Omron CX-Programmer project NewProject (CX-Programmer 7.21)

# PLC NewPLC1: CJ1M CPU13
I/O table (CPU CJ1M-CPU13): rack 0 slot 0 CJ1W-SCU41-V1

## Global symbols (name address type ; comment)
D0 CHANNEL  ; Ctrl1
D1 CHANNEL  ; Ctrl2
D10 CHANNEL  ; Send Word
D20 CHANNEL  ; No. To Send
D30 CHANNEL  ; Receive Word
D40 CHANNEL  ; No. To Receive
D70 CHANNEL  ; Batt
D71 CHANNEL  ; Sgn1
D72 CHANNEL  ; Dig1
D73 CHANNEL  ; Sgn2
D74 CHANNEL  ; Dig2
D75 CHANNEL  ; ID
D76 CHANNEL  ; Disp1
D77 CHANNEL  ; Dly
D78 CHANNEL  ; StpSgn
D79 CHANNEL  ; RunSgn
D80 CHANNEL  ; FinSgn
D81 CHANNEL  ; RsdSgn
D82 CHANNEL  ; Disp2
D83 CHANNEL  ; Err
D84 CHANNEL  ; Page
D85 CHANNEL  ; FileNo.
D86 CHANNEL  ; ErrNo.
D87 CHANNEL  ; DataNo.2
D88 CHANNEL  ; DataNo.1 LSB
D89 CHANNEL  ; MsdErr
D90 CHANNEL  ; MemSgn
D92 CHANNEL  ; DataNo.2 MSB
D93 CHANNEL  ; DataNo.

## Program NewProgram1 (cyclic task 0)

### Section Section1

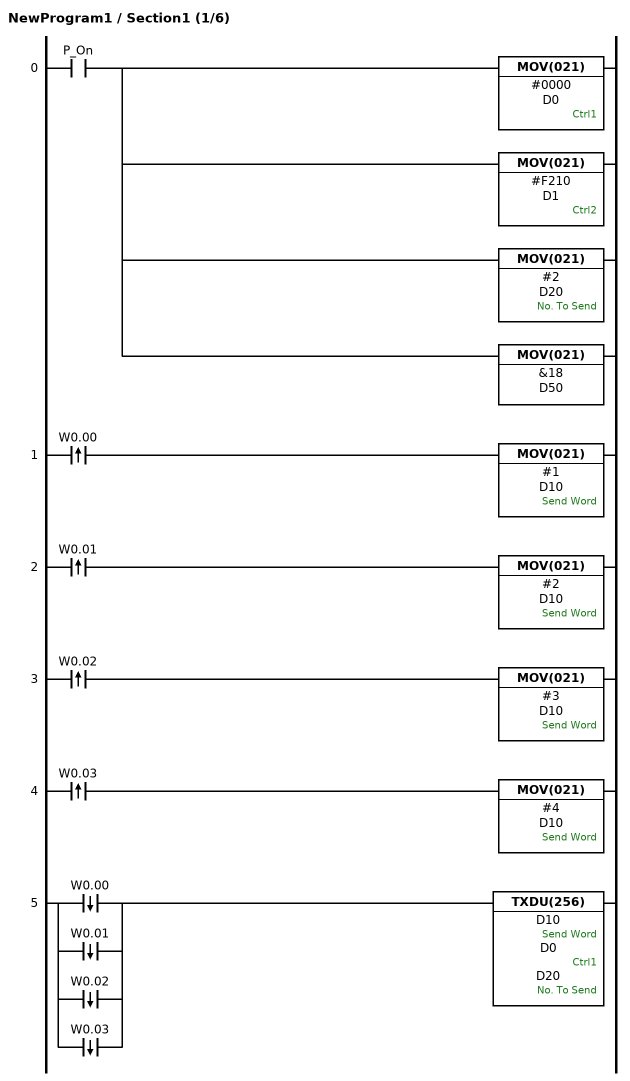
; rung 0
LD P_On
MOV(021) #0000 D0  ; Ctrl1
MOV(021) #F210 D1  ; Ctrl2
MOV(021) #2 D20  ; No. To Send
MOV(021) &18 D50
; rung 1
@LD W0.00
MOV(021) #1 D10  ; Send Word
; rung 2
@LD W0.01
MOV(021) #2 D10  ; Send Word
; rung 3
@LD W0.02
MOV(021) #3 D10  ; Send Word
; rung 4
@LD W0.03
MOV(021) #4 D10  ; Send Word
; rung 5
%LD W0.00
%OR W0.01
%OR W0.02
%OR W0.03
TXDU(256) D10 D0 D20  ; Send Word, Ctrl1, No. To Send

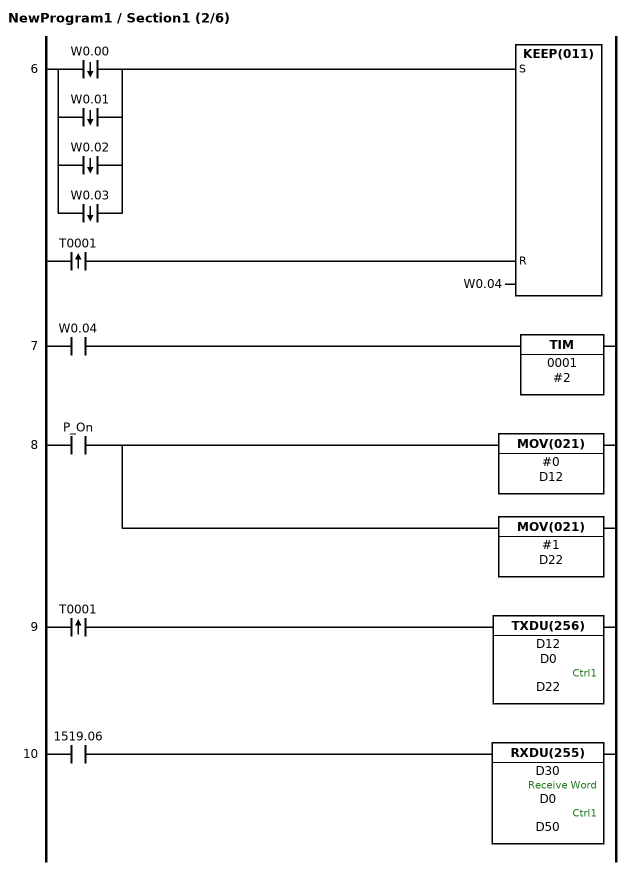
; rung 6
%LD W0.00
%OR W0.01
%OR W0.02
%OR W0.03
@LD T0001
KEEP(011) W0.04
; rung 7
LD W0.04
TIM 0001 #2
; rung 8
LD P_On
MOV(021) #0 D12
MOV(021) #1 D22
; rung 9
@LD T0001
TXDU(256) D12 D0 D22  ; Ctrl1
; rung 10
LD 1519.06
RXDU(255) D30 D0 D50  ; Receive Word, Ctrl1

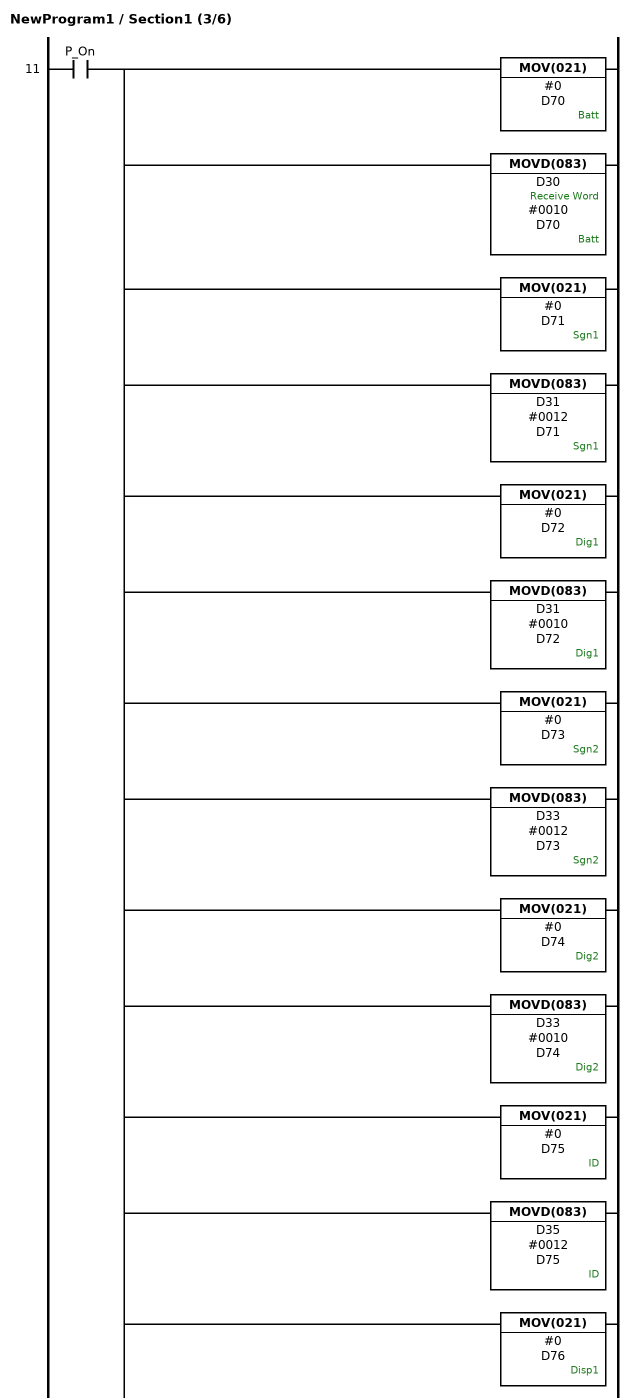

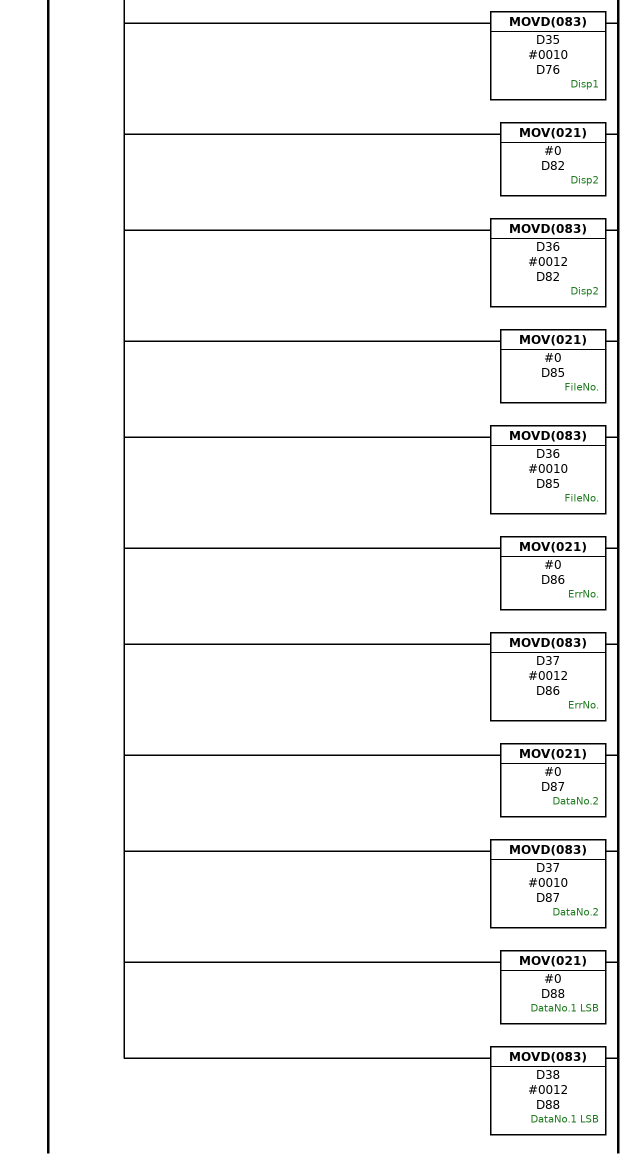
; rung 11
LD P_On
MOV(021) #0 D70  ; Batt
MOVD(083) D30 #0010 D70  ; Receive Word, Batt
MOV(021) #0 D71  ; Sgn1
MOVD(083) D31 #0012 D71  ; Sgn1
MOV(021) #0 D72  ; Dig1
MOVD(083) D31 #0010 D72  ; Dig1
MOV(021) #0 D73  ; Sgn2
MOVD(083) D33 #0012 D73  ; Sgn2
MOV(021) #0 D74  ; Dig2
MOVD(083) D33 #0010 D74  ; Dig2
MOV(021) #0 D75  ; ID
MOVD(083) D35 #0012 D75  ; ID
MOV(021) #0 D76  ; Disp1
MOVD(083) D35 #0010 D76  ; Disp1
MOV(021) #0 D82  ; Disp2
MOVD(083) D36 #0012 D82  ; Disp2
MOV(021) #0 D85  ; FileNo.
MOVD(083) D36 #0010 D85  ; FileNo.
MOV(021) #0 D86  ; ErrNo.
MOVD(083) D37 #0012 D86  ; ErrNo.
MOV(021) #0 D87  ; DataNo.2
MOVD(083) D37 #0010 D87  ; DataNo.2
MOV(021) #0 D88  ; DataNo.1 LSB
MOVD(083) D38 #0012 D88  ; DataNo.1 LSB

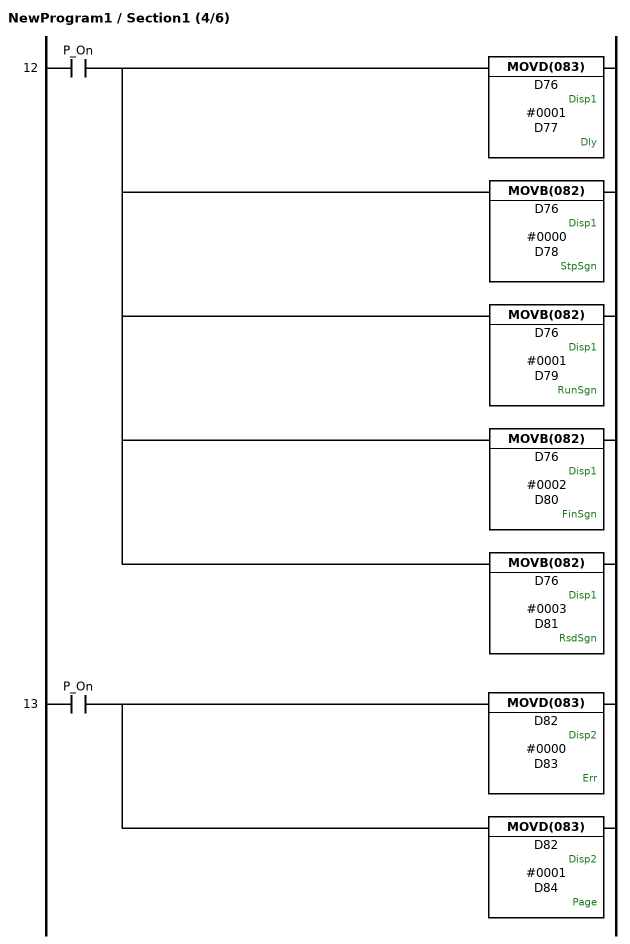
; rung 12
LD P_On
MOVD(083) D76 #0001 D77  ; Disp1, Dly
MOVB(082) D76 #0000 D78  ; Disp1, StpSgn
MOVB(082) D76 #0001 D79  ; Disp1, RunSgn
MOVB(082) D76 #0002 D80  ; Disp1, FinSgn
MOVB(082) D76 #0003 D81  ; Disp1, RsdSgn
; rung 13
LD P_On
MOVD(083) D82 #0000 D83  ; Disp2, Err
MOVD(083) D82 #0001 D84  ; Disp2, Page

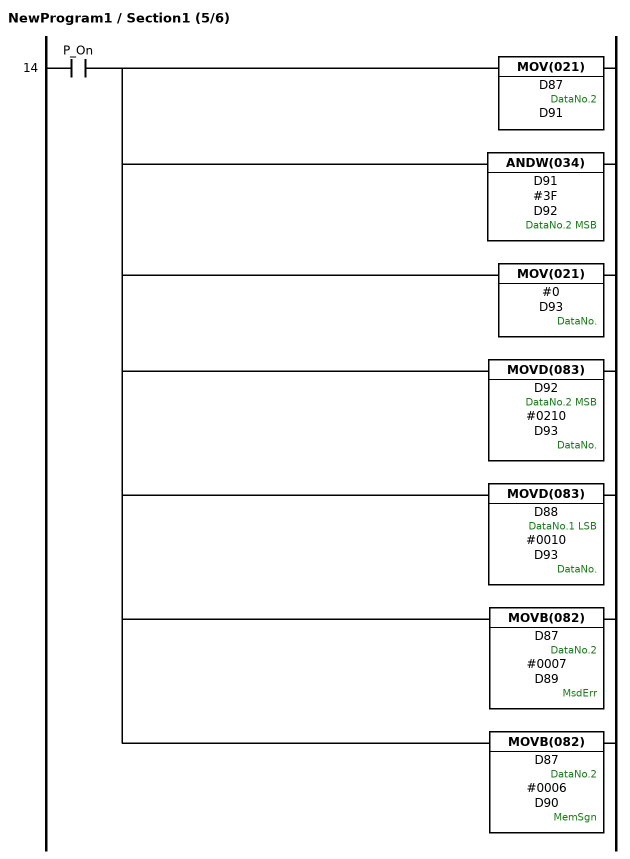
; rung 14
LD P_On
MOV(021) D87 D91  ; DataNo.2
ANDW(034) D91 #3F D92  ; DataNo.2 MSB
MOV(021) #0 D93  ; DataNo.
MOVD(083) D92 #0210 D93  ; DataNo.2 MSB, DataNo.
MOVD(083) D88 #0010 D93  ; DataNo.1 LSB, DataNo.
MOVB(082) D87 #0007 D89  ; DataNo.2, MsdErr
MOVB(082) D87 #0006 D90  ; DataNo.2, MemSgn

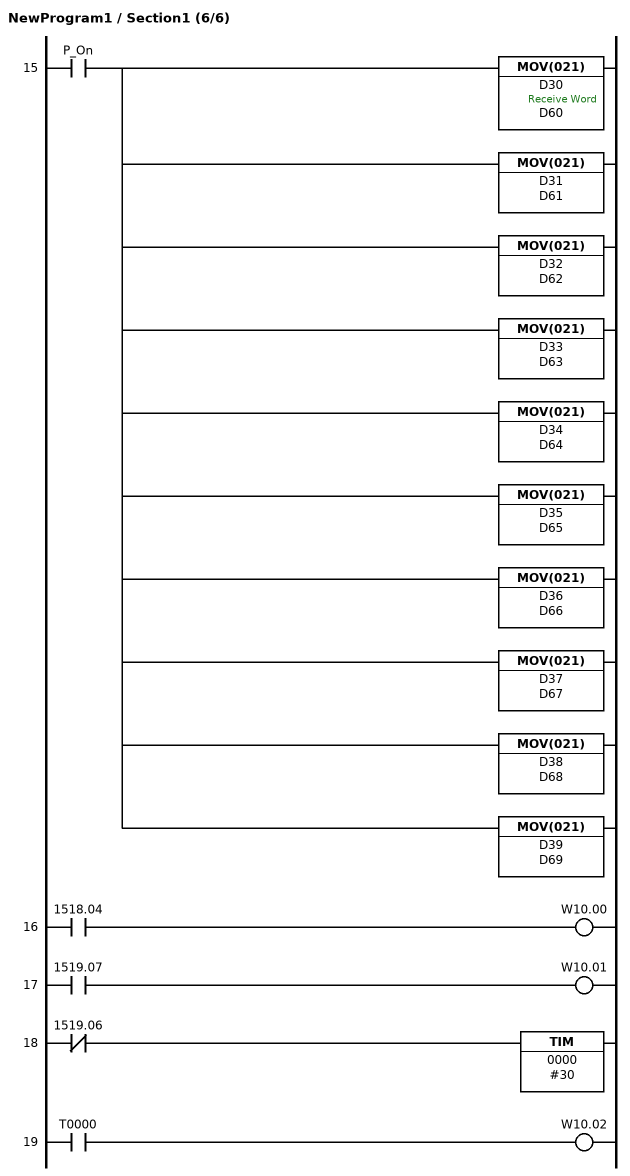
; rung 15
LD P_On
MOV(021) D30 D60  ; Receive Word
MOV(021) D31 D61
MOV(021) D32 D62
MOV(021) D33 D63
MOV(021) D34 D64
MOV(021) D35 D65
MOV(021) D36 D66
MOV(021) D37 D67
MOV(021) D38 D68
MOV(021) D39 D69
; rung 16
LD 1518.04
OUT W10.00
; rung 17
LD 1519.07
OUT W10.01
; rung 18
LDNOT 1519.06
TIM 0000 #30
; rung 19
LD T0000
OUT W10.02

### Section END
; rung 0
END(001)